{attribute 'qualified_only'}
{attribute 'strict'}
TYPE E_STM_STEP :
(
	resetEnv := 0,
	computeAction,
	executeAction,
	updateQtable,
	trackReward,
	updateState,
	checkIfDone
);
END_TYPE

(* stored: Version 1.1.0.1, ProductVersion 3.1.4024.12
   DUT E_STM_STEP: Id {6a806c30-b009-46d4-9b9a-63b56b93c40a} *)
